DATA_BLOCK "dbArchiveAutoDoor"
{ S7_Optimized_Access := 'TRUE' }
VERSION : 0.8
NON_RETAIN
"fbArchiveAutoDoor"

BEGIN

END_DATA_BLOCK

